Yaskawa INFORM job: HOME_POS_ST.JBI

/JOB
//NAME HOME_POS_ST
//POS
///NPOS 1,0,0,0,0,0
///TOOL 0
///POSTYPE PULSE
///PULSE
C00000=142529,-8517,3701,5795,-74419,-9941
//INST
///DATE 2021/10/11 09:29
///ATTR SC,RW
///GROUP1 RB1
NOP
MOVJ C00000
END
